(* CODESYS project Read_Basic_Info.export

Project tree, tasks and I/O mapping:
  program Read_Basic_Info [ST]
*)

// Read_Basic_Info
PROGRAM Read_Basic_Info
VAR	
	// read cfg message
	ReadCfg : ArcaLibrary.SYS_GetConfigInfo;
END_VAR

// read how many axis has been config
ReadCfg(axisnumber => Num_of_Axis_GV, groupnumber => Num_of_Groups_GV, cameranumber => Num_of_Cams_GV
	, MotionCfgOk => MotionCfgOK_GV, ecatcfgok => ECatCfgOk_GV, visioncfgok => VisionCfgOk_GV);

END_PROGRAM
